{attribute 'linkalways'} 
{attribute 'no_explicit_call' := 'This FB is a CLASS and must be accessed using methods or properties'}
{attribute 'enable_dynamic_creation'}
FUNCTION_BLOCK FINAL SUB_REAL EXTENDS Node
VAR
	in1 : _REAL(0.0);
	in2 : _REAL(0.0);
	out : _REAL(0.0);
END_VAR

METHOD PUBLIC Clone : I_Node
VAR
	pNode : POINTER TO SUB_REAL;
END_VAR
pNode := __NEW(SUB_REAL);
Clone := pNode^;
END_METHOD

METHOD FB_init : BOOL
VAR_INPUT
	bInitRetains : BOOL; // if TRUE, the retain variables are initialized (warm start / cold start)
	bInCopyCode : BOOL;  // if TRUE, the instance afterwards gets moved into the copy code (online change)
END_VAR
AddInput('in1',THIS^.in1);
AddInput('in2',THIS^.in2);
AddOutput('out', THIS^.out);
END_METHOD

METHOD PROTECTED OnExecute
VAR
END_VAR
out.Value := in1.Value - in2.Value;
END_METHOD

END_FUNCTION_BLOCK

(* stored: Version 1.1.0.1, ProductVersion 3.1.4024.15
   POU SUB_REAL: Id {d92eaa57-5537-4a66-a41b-f07423be942b}, SpecialFunc None
   Folder Constructor: Id {a5c85a15-20ba-4149-8ea1-0a6aa64d4b11}
   Method Clone: Id {83ff7d97-6912-4eaa-b317-f8b7096ee7be}
   Method FB_init: Id {1dfd9738-0ea3-4919-b46a-1f74ebf0d9ed}
   Method OnExecute: Id {05a75555-8856-4044-bbcb-ba4767169d8e} *)
